{attribute 'GeneratedUsingTerminal: EJ9576-0000-0022'}
{attribute addProperty BoxType "EJ9576-0000-0022"}
{attribute addProperty Description "EJ9576 Brake chopper terminal"}
{attribute addProperty Physics "KK"}
{attribute addProperty Id "BCT_InputsAT %I*BCT_Inputs_7ACE8FA617WcStateAT %I*WcState_9091E0EB2InfoDataAT %I*InfoData_32EB74EA10"}
{attribute addProperty CRC "3290514118"}
{attribute addProperty Size "29"}
TYPE EJ9576_C42142C6 EXTENDS EtcSlaveTerminalBase_947E5A46 :
STRUCT
	{attribute addProperty Name "BCT_Inputs"}
	BCT_Inputs : BCT_Inputs_7ACE8FA6;
	{attribute addProperty Name "WcState"}
	WcState : WcState_9091E0EB;
	{attribute addProperty Name "InfoData"}
	InfoData : InfoData_32EB74EA;
END_STRUCT
END_TYPE

(* stored: Version 1.2.0.0, ProductVersion 3.1.4024.11
   DUT EJ9576_C42142C6: Id {894ac510-1a83-4613-8b07-2c13f13942f7} *)
